ABB RobotStudio station: EstaciónDeSoldadura_20200720-180749.rsstn

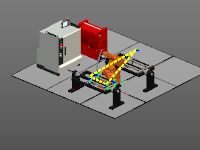
Station EstaciónDeSoldadura (saved by RobotStudio 7.0.8746.631)
Controller IRB_140_6kg_0.81m
  mechanical unit ROB_1: IRB140_6_81_C_03, 6 joints, base frame (0, 0, 0) mm
Layout (positions relative to the parent item):
  - IRB140_6_81_C_03 [mechanism, from Robots\IRB140_6_81_C_G_03.rslib] at (0, 0, 0) mm; joint values [-1.8783, -0.6506, -0.0242, -2.886, -1.3303, 2.8958] (rad or m)
  - AW_Gun_PSF_25 [mechanism, from Tools\AW_Gun_PSF_25.rslib] at (-45, -194.41, 837.83) mm, rotated rx 180 ry 54.2 rz 90 deg
  - IRC5_Singel-Cabinet [part, from Equipment\IRC5_Singel-Cabinet.rslib] at (-1350, 0, 100) mm, rotated rx 90 ry 0 rz 90 deg
  - Fronius_TPS4000_rev0 [part, from Equipment\Fronius_TPS4000.rslib] at (-1350, 900, 0) mm, rotated rx 0 ry 0 rz -90 deg
  - FlexPendant [part, from Equipment\FlexPendant.rslib] at (-1350, 0, 1100) mm, rotated rx 0 ry 0 rz 90 deg
  - Mesa [mechanism] at (-540, -540, 0) mm; joint values [0] (rad or m)
      links: L1, L2, L3
  - Mesa_2 [mechanism] at (-540, 540, 0) mm; joint values [0] (rad or m)
      links: L1, L2, L3
Attachment: AW_Gun_PSF_25 is attached to IRB140_6_81_C_03 / Link6
Attachment: Workobject_Mesa1 is attached to Mesa / L2
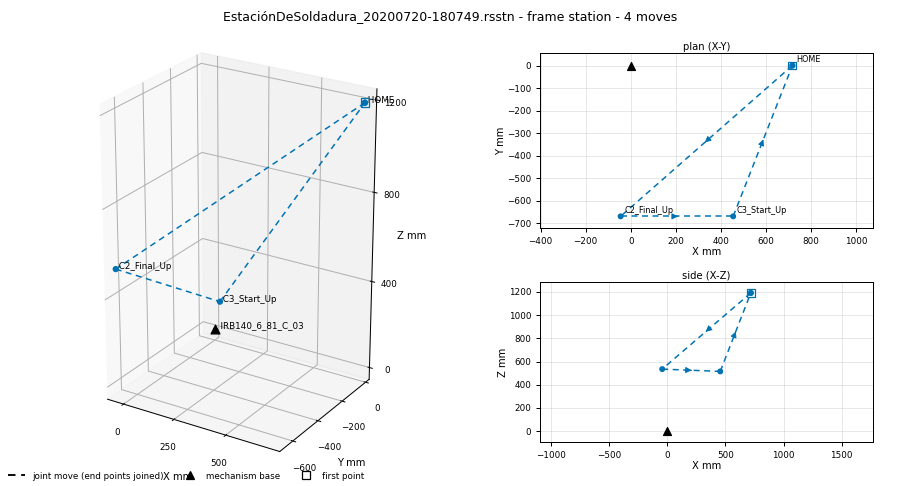
[picture p0: tool path of EstaciónDeSoldadura_20200720-180749.rsstn in frame station, 4 of 4 moves have a stored position in this frame; points joined in program order, loops and branches not executed]
Targets, tools, work objects and paths stored in the station, written as RAPID:
! task T_ROB1
MODULE CalibData
  PERS tooldata AW_Gun:=[TRUE,[[119.5,0,352],[0.890213743,0,0.455543074,0]],[1,[0,0,100],[1,0,0,0],0,0,0]];
  PERS wobjdata Workobject_Mesa1:=[FALSE,TRUE,"",[[-590,-540,370],[0.707106781,0.707106781,0,0]],[[0,0,0],[1,0,0,0]]];
ENDMODULE

! task T_ROB1
MODULE Module1
  CONST robtarget C1_Start:=[[545,65,-130],[0.5,0.5,0.5,-0.5],[-2,-2,1,1],[9E+09,9E+09,9E+09,9E+09,9E+09,9E+09]];
  CONST robtarget C1_Final:=[[545,65,-100],[0.5,0.5,0.5,-0.5],[-2,-2,1,1],[9E+09,9E+09,9E+09,9E+09,9E+09,9E+09]];
  CONST robtarget C2_Start:=[[545,65,100],[0.5,0.5,0.5,-0.5],[-2,-2,1,1],[9E+09,9E+09,9E+09,9E+09,9E+09,9E+09]];
  CONST robtarget C2_Final:=[[545,65,130],[0.5,0.5,0.5,-0.5],[-2,-2,1,1],[9E+09,9E+09,9E+09,9E+09,9E+09,9E+09]];
  CONST robtarget C3_Start:=[[1045,65,130],[0.5,0.5,0.5,-0.5],[0,0,0,0],[9E+09,9E+09,9E+09,9E+09,9E+09,9E+09]];
  CONST robtarget C3_Final:=[[1045,65,100],[0.5,0.5,0.5,-0.5],[0,0,0,0],[9E+09,9E+09,9E+09,9E+09,9E+09,9E+09]];
  CONST robtarget C4_Start:=[[1045,65,-100],[0.5,0.5,0.5,-0.5],[0,0,0,0],[9E+09,9E+09,9E+09,9E+09,9E+09,9E+09]];
  CONST robtarget C4_Final:=[[1045,65,-130],[0.5,0.5,0.5,-0.5],[0,0,0,0],[9E+09,9E+09,9E+09,9E+09,9E+09,9E+09]];
  CONST robtarget C1_Final_Up:=[[545,165,-100],[0.5,0.5,0.5,-0.5],[-2,-2,1,1],[9E+09,9E+09,9E+09,9E+09,9E+09,9E+09]];
  CONST robtarget C1_Start_Up:=[[545,165,-130],[0.5,0.5,0.5,-0.5],[-2,-2,1,1],[9E+09,9E+09,9E+09,9E+09,9E+09,9E+09]];
  CONST robtarget C2_Final_Up:=[[545,165,130],[0.5,0.5,0.5,-0.5],[-2,-2,1,1],[9E+09,9E+09,9E+09,9E+09,9E+09,9E+09]];
  CONST robtarget C2_Start_Up:=[[545,165,100],[0.5,0.5,0.5,-0.5],[-2,-2,1,1],[9E+09,9E+09,9E+09,9E+09,9E+09,9E+09]];
  CONST robtarget C3_Final_Up:=[[1045,165,100],[0.5,0.5,0.5,-0.5],[0,0,0,0],[9E+09,9E+09,9E+09,9E+09,9E+09,9E+09]];
  CONST robtarget C3_Start_Up:=[[1045,145,130],[0.5,0.5,0.5,-0.5],[-1,-1,0,0],[9E+09,9E+09,9E+09,9E+09,9E+09,9E+09]];
  CONST robtarget C4_Final_Up:=[[1045,165,-130],[0.5,0.5,0.5,-0.5],[0,0,0,0],[9E+09,9E+09,9E+09,9E+09,9E+09,9E+09]];
  CONST robtarget C4_Start_Up:=[[1045,165,-100],[0.5,0.5,0.5,-0.5],[0,0,0,0],[9E+09,9E+09,9E+09,9E+09,9E+09,9E+09]];
  CONST robtarget C5_Start:=[[545,35,130],[0.5,-0.5,-0.5,-0.5],[0,0,0,0],[9E+09,9E+09,9E+09,9E+09,9E+09,9E+09]];
  CONST robtarget C5_Final:=[[545,35,100],[0.5,-0.5,-0.5,-0.5],[0,0,0,0],[9E+09,9E+09,9E+09,9E+09,9E+09,9E+09]];
  CONST robtarget C6_Start:=[[545,35,-100],[0.5,-0.5,-0.5,-0.5],[0,0,0,0],[9E+09,9E+09,9E+09,9E+09,9E+09,9E+09]];
  CONST robtarget C6_Final:=[[545,35,-130],[0.5,-0.5,-0.5,-0.5],[0,0,0,0],[9E+09,9E+09,9E+09,9E+09,9E+09,9E+09]];
  CONST robtarget C7_Start:=[[1045,35,-130],[0.5,-0.5,-0.5,-0.5],[0,0,0,0],[9E+09,9E+09,9E+09,9E+09,9E+09,9E+09]];
  CONST robtarget C7_Final:=[[1045,35,-100],[0.5,-0.5,-0.5,-0.5],[0,0,0,0],[9E+09,9E+09,9E+09,9E+09,9E+09,9E+09]];
  CONST robtarget C8_Start:=[[1045,35,100],[0.5,-0.5,-0.5,-0.5],[0,0,0,0],[9E+09,9E+09,9E+09,9E+09,9E+09,9E+09]];
  CONST robtarget C8_Final:=[[1045,35,130],[0.5,-0.5,-0.5,-0.5],[0,0,0,0],[9E+09,9E+09,9E+09,9E+09,9E+09,9E+09]];
  CONST robtarget C5_Final_Up:=[[545,-65,100],[0.5,-0.5,-0.5,-0.5],[0,0,0,0],[9E+09,9E+09,9E+09,9E+09,9E+09,9E+09]];
  CONST robtarget C5_Start_Up:=[[545,-65,130],[0.5,-0.5,-0.5,-0.5],[0,0,0,0],[9E+09,9E+09,9E+09,9E+09,9E+09,9E+09]];
  CONST robtarget C6_Final_Up:=[[545,-65,-130],[0.5,-0.5,-0.5,-0.5],[0,0,0,0],[9E+09,9E+09,9E+09,9E+09,9E+09,9E+09]];
  CONST robtarget C6_Start_Up:=[[545,-65,-100],[0.5,-0.5,-0.5,-0.5],[0,0,0,0],[9E+09,9E+09,9E+09,9E+09,9E+09,9E+09]];
  CONST robtarget C7_Final_Up:=[[1045,-65,-100],[0.5,-0.5,-0.5,-0.5],[0,0,0,0],[9E+09,9E+09,9E+09,9E+09,9E+09,9E+09]];
  CONST robtarget C7_Start_Up:=[[1045,-65,-130],[0.5,-0.5,-0.5,-0.5],[0,0,0,0],[9E+09,9E+09,9E+09,9E+09,9E+09,9E+09]];
  CONST robtarget C8_Final_Up:=[[1045,-65,130],[0.5,-0.5,-0.5,-0.5],[0,0,0,0],[9E+09,9E+09,9E+09,9E+09,9E+09,9E+09]];
  CONST robtarget C8_Start_Up:=[[1045,-65,100],[0.5,-0.5,-0.5,-0.5],[0,0,0,0],[9E+09,9E+09,9E+09,9E+09,9E+09,9E+09]];
  CONST robtarget HOME:=[[1308.063364957,821.064844254,-540],[0.458291086,-0.458291086,0.538487958,-0.538487958],[0,0,0,0],[9E+09,9E+09,9E+09,9E+09,9E+09,9E+09]];
  PROC BOCARRIBA_1()
    MoveJ HOME,v1000,z100,AW_Gun\WObj:=Workobject_Mesa1;
    MoveJ C2_Final_Up,v1000,z100,AW_Gun\WObj:=Workobject_Mesa1;
    MoveJ C3_Start_Up,v200,z100,AW_Gun\WObj:=Workobject_Mesa1;
    MoveJ HOME,v1000,z100,AW_Gun\WObj:=Workobject_Mesa1;
  ENDPROC
  PROC main()
    BOCARRIBA_1;
  ENDPROC
ENDMODULE

